FUNCTION_BLOCK F_SUB_DT_DT (* Subtracts two time data types *)
  (* Standard: 61131-3; Classification: Arithmetic; Function: SUBTRACTOR; Type: Mathematical function *)
  (* Version 1.0, 2013-09-10, 4DIAC-IDE, 4DIAC-Consortium *)
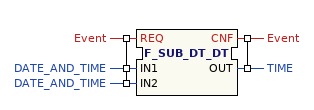
  EVENT_INPUT
    REQ WITH IN1, IN2; (* Normal Execution Request *)
  END_EVENT
  EVENT_OUTPUT
    CNF WITH OUT; (* Execution Confirmation *)
  END_EVENT
  VAR_INPUT
    IN1 : DATE_AND_TIME; (* First funtion input *)
    IN2 : DATE_AND_TIME; (* Second function input *)
  END_VAR
  VAR_OUTPUT
    OUT : TIME; (* Function output *)
  END_VAR
END_FUNCTION_BLOCK
